SUBAPPLICATION Uebung_034 (* Analog-Eingang auf PWM Ausgang *)
  (* Standard: 61499-2; Description: Copyright (c) 2023 Meisterschulen am Ostbahnhof This program and the accompanying materials are made available under the terms of the Eclipse Public License 2.0 which is available at https://www.eclipse.org/legal/epl-2.0/ SPDX-License-Identifier: EPL-2.0 *)
  (* Version 1.0, 2023-10-23, Franz Höpfinger, Meisterschulen am Ostbahnhof *)
  IMPORT logiBUS::io::AI::logiBUS_AI;
  IMPORT logiBUS::io::DQ::logiBUS_DO::Output_Q4;
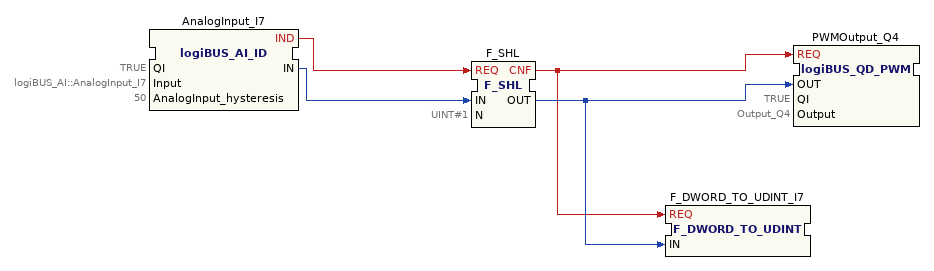
  FBS
    AnalogInput_I7 : logiBUS::io::AI::logiBUS_AI_ID(QI := TRUE, Input := logiBUS_AI::AnalogInput_I7, AnalogInput_hysteresis := 50);
    F_DWORD_TO_UDINT_I7 : iec61131::conversion::F_DWORD_TO_UDINT;
    PWMOutput_Q4 : logiBUS::io::DQ::logiBUS_QD_PWM(QI := TRUE, Output := Output_Q4);
    F_SHL : iec61131::bitwiseOperators::F_SHL(N := UINT#1);
  END_FBS
  EVENT_CONNECTIONS
    AnalogInput_I7.IND TO F_SHL.REQ;
    F_SHL.CNF TO F_DWORD_TO_UDINT_I7.REQ;
    F_SHL.CNF TO PWMOutput_Q4.REQ;
  END_CONNECTIONS
  DATA_CONNECTIONS
    AnalogInput_I7.IN TO F_SHL.IN;
    F_SHL.OUT TO PWMOutput_Q4.OUT;
    F_SHL.OUT TO F_DWORD_TO_UDINT_I7.IN;
  END_CONNECTIONS
END_SUBAPPLICATION
